(* IEC 61131-3 sources: repolevel_ST_code_completion/output/0121完整版本/repoeval_Proxy_Application/readful_result, 2 files *)

(* ---- Proxy.st ---- *)
{attribute 'enable_dynamic_creation'}
FUNCTION_BLOCK Proxy IMPLEMENTS  Subject_Interface
VAR_INPUT
END_VAR
VAR_OUTPUT
END_VAR
VAR
	refToRealSubject : POINTER TO Realsubject;
	iTempPassword : INT;
END_VAR
VAR_STAT
	iRealPassword : INT := 1234;
END_VAR

METHOD fb_init: BOOL
// The fb_init METHOD is implemented outside of variable declarations
// Reusing declared variables, eliminating invalid `VAR` blocks.

IF refToRealSubject <> 0 THEN
  // Assuming refToRealSubject is initialized elsewhere
  iTempPassword := iRealPassword; // Use declared variables directly
  RETURN(TRUE);
END_IF;

IF iTempPassword = iRealPassword THEN
  IF bReadWrite THEN
    // Simulated behavior using declared variables
    iTempPassword := iSetValue;
  ELSE
    iSetValue := iTempPassword; // Example substitution for refToRealSubject^.iProp
  END_IF;
END_IF;

RETURN(TRUE); // Indicate successful operation
END_METHOD
END_FUNCTION_BLOCK

(* ---- Realsubject.st ---- *)
{attribute 'enable_dynamic_creation'}
FUNCTION_BLOCK Realsubject IMPLEMENTS  Subject_Interface
VAR_INPUT
END_VAR
VAR_OUTPUT
END_VAR
VAR
    // Variable to get and set values
    iProp: INT;
END_VAR

VAR_STAT
    // No static variables required for this implementation
END_VAR

// Declaration of public methods before starting the implementation part

// Declare and implement methods properly

// Proper separation of method declarations and implementations

 METHOD Get_Method : INT
 // Declaration of method Get_Method
 END_METHOD

 METHOD IMPLEMENTATION Get_Method
 // Implementation of Get_Method
 Get_Method := iProp; // Return the value of iProp
 END_METHOD

 METHOD Set_Method
 VAR_INPUT
  num : INT; // Value to be set on the iProp variable
 END_VAR
 // Declaration of method Set_Method
 END_METHOD

 METHOD IMPLEMENTATION Set_Method
 // Implementation of Set_Method
 iProp := num; // Assign the value of num to iProp
 END_METHOD
END_FUNCTION_BLOCK
